TYPE g_ttrrr:
    STRUCT
        field1: g_trr;
        field2: LREAL;
    END_STRUCT
END_TYPE

(* stored: ProductVersion 3.1.0.18, Version 1.1.0.1 *)
